(* CoDeSys 2.3.9.50 project: Test.pro *)
(* Libraries: STANDARD.LIB 5.6.98 12:03:02 *)

(* Task configuration *)
TASK Standard (PRIORITY := 0, INTERVAL := T#10ms);
	MAIN
END_TASK

(* POU MAIN, ST *)
PROGRAM MAIN
VAR
	InMainVolt AT %IX0.0 : BOOL;
	OutMainVolt AT %QX0.0 : BOOL;

	In0_1 AT %IX0.1 : BOOL;
	In0_2 AT %IX0.2 : BOOL;
	In0_3 AT %IX0.3 : BOOL;
	In0_4 AT %IX0.4 : BOOL;
	In0_5 AT %IX0.5 : BOOL;
	In0_6 AT %IX0.6 : BOOL;
	In0_7 AT %IX0.7 : BOOL;
	In0_8 AT %IX0.8 : BOOL;

	Out0_1 AT %QX0.1 : BOOL;
	Out0_2 AT %QX0.2 : BOOL;
	Out0_3 AT %QX0.3 : BOOL;
	Out0_4 AT %QX0.4 : BOOL;
	Out0_5 AT %QX0.5 : BOOL;
	Out0_6 AT %QX0.6 : BOOL;
	Out0_7 AT %QX0.7 : BOOL;
	Out0_8 AT %QX0.8 : BOOL;


	In1_1 AT %IX0.9 : BOOL;
	In1_2 AT %IX0.10 : BOOL;
	In1_3 AT %IX0.11 : BOOL;
	In1_4 AT %IX0.12 : BOOL;
	In1_5 AT %IX0.13 : BOOL;
	In1_6 AT %IX0.14 : BOOL;
	In1_7 AT %IX0.15 : BOOL;
	In1_8 AT %IX0.16 : BOOL;

	Out1_1 AT %QX0.9 : BOOL;
	Out1_2 AT %QX0.10 : BOOL;
	Out1_3 AT %QX0.11 : BOOL;
	Out1_4 AT %QX0.12 : BOOL;
	Out1_5 AT %QX0.13 : BOOL;
	Out1_6 AT %QX0.14 : BOOL;
	Out1_7 AT %QX0.15 : BOOL;
	Out1_8 AT %QX0.16 : BOOL;


	In2_1 AT %IX0.17 : BOOL;
	In2_2 AT %IX0.18 : BOOL;
	In2_3 AT %IX0.19 : BOOL;
	In2_4 AT %IX0.20 : BOOL;
	In2_5 AT %IX0.21 : BOOL;
	In2_6 AT %IX0.22 : BOOL;
	In2_7 AT %IX0.23 : BOOL;
	In2_8 AT %IX0.24 : BOOL;

	Out2_1 AT %QX0.17 : BOOL;
	Out2_2 AT %QX0.18 : BOOL;
	Out2_3 AT %QX0.19 : BOOL;
	Out2_4 AT %QX0.20 : BOOL;
	Out2_5 AT %QX0.21 : BOOL;
	Out2_6 AT %QX0.22 : BOOL;
	Out2_7 AT %QX0.23 : BOOL;
	Out2_8 AT %QX0.24 : BOOL;

END_VAR
(* init *)
IF InMainVolt THEN
	OutMainVolt := TRUE ;
END_IF
END_PROGRAM
